PROGRAM P_FlowControl
VAR
	fbFlowControlMain : FB_FlowControl;
	fbFlowControlJib : FB_FlowControl;
END_VAR

// 
// 
// fbFlowControlMain(
// 	fArea1 := G_Parameters.fAreaMain,
// 	fArea2 := G_Parameters.fAreaJib,
// 	fFlow1 := G_OPC.fMainFlowA,
// 	fFlow2 := G_OPC.fJibFlowA,
// 	bEqualSpeed := TRUE,
// 	
// 	fSpeedRef1 => G_OPC.fFlowTest1,
// 	fSpeedRef2 => G_OPC.fFlowTest2
// );
//

END_PROGRAM

(* stored: Version 1.1.0.1
   POU P_FlowControl: Id {02257286-ea62-4045-8238-7992179f10c6}, SpecialFunc None *)
